//{attribute 'qualified_only'}
VAR_GLOBAL
	
//	r_Accelerator_Setpoint	: REAL := 1E-12; (*unrealistic setpoint currently*)
	{attribute 'pytmc' := 'pv: TMO:FEE:VAC:OVRDON'}
	xSystemOverrideMode_FEE	: BOOL := FALSE; (* Global system override for the TMO FEE Vacuum System *)
	
	{attribute 'pytmc' := 'pv: TMO:NEH:VAC:OVRDON'}
	xSystemOverrideMode_TMO	: BOOL := FALSE; (* Global system override for the TMO hutch Vacuum System *)
	
	{attribute 'pytmc' := 'pv: TMO:NEH:TURBO:FAULT'}
	xTurboFault: BOOL := FALSE; (* True if any hutch turbo is not at speed or fault *)	
	
	{attribute 'pytmc' := 'pv: TMO:NEH:VALVE:FAULT'}
	xValveFault: BOOL := FALSE; (* True if any hutch turbo is not at speed or fault *)	
END_VAR

(* stored: Version 1.1.0.1, ProductVersion 3.1.4022.18
   GVL GVL_Variables: Id {0b31be2f-6c9a-4798-a48f-4b64605f971e} *)
